PROGRAM HMIHelper
VAR
	HMI_XTSMoverInfo	: ARRAY[1..10] OF HMI_XTSMoverInfo_typ;
	i					: INT;
	Init				: BOOL;
END_VAR

IF NOT Init THEN
	FOR i := 1 TO (SIZEOF(HMI_XTSMoverInfo) / SIZEOF(HMI_XTSMoverInfo[1])) DO
		HMI_XTSMoverInfo[i].Index	:= i;
	END_FOR
	Init	:= TRUE;
END_IF

FOR i := 1 TO (SIZEOF(HMI_XTSMoverInfo) / SIZEOF(HMI_XTSMoverInfo[1])) DO
	HMI_XTSMoverInfo[i].Ready		:= Main.XTS.Mover[i].Ready;
	HMI_XTSMoverInfo[i].Position	:= Main.XTS.Mover[i].TrackInfo.TrackPosition;
END_FOR

END_PROGRAM

(* stored: Version 1.1.0.1, ProductVersion 3.1.4026.12
   POU HMIHelper: Id {86407be7-6f6a-0ed9-2497-dafead09aa63}, SpecialFunc None *)
